(* PLC project Untitled2, Machine Expert Logic Builder V22.1.1.0, author vboxuser *)
(* stored: creationDateTime 2026-02-09T20:32:05.1605517, version 0.0.0.0, modificationDateTime 2026-02-09T20:28:06.3101652 *)

FUNCTION_BLOCK FB_Example
  VAR CONSTANT
    cArrSize : INT := 100;
  END_VAR
  VAR
    values : ARRAY[1..cArrSize] OF REAL;
    count : INT := 0;
  END_VAR

            
          

METHOD AddValue
  VAR_INPUT
    value : REAL;
  END_VAR
  VAR
    i : INT;
  END_VAR
                  IF THIS^.count < THIS^.cArrSize THEN
    THIS^.count := THIS^.count + 1;
    THIS^.values[THIS^.count] := value;
ELSE
	(*Handle overflow, move array up 1 step and add new value as the newest value *)
     FOR i := 1 TO THIS^.cArrSize - 1 DO
         THIS^.values[i] := THIS^.values[i + 1];
     END_FOR
     
     values[THIS^.cArrSize] := value;
     THIS^.count := THIS^.cArrSize;
END_IF
                
END_METHOD

PROPERTY GetCount : INT
GET
                    GetCount := THIS^.count;
                  
END_GET
END_PROPERTY
END_FUNCTION_BLOCK
